// TwinCAT 3 PLC project MRA_LIB
// Title: MRA_LIB
// Company: MRA Solutions
// ProjectVersion: 1.0.5
// ProgramVersion: 3.1.4023.0
// libraries:
//   Tc2_EIB, * (Beckhoff Automation GmbH)
//   Tc2_IoFunctions, * (Beckhoff Automation GmbH)
//   Tc2_ModbusRTU, * (Beckhoff Automation GmbH)
//   Tc2_Standard, * (Beckhoff Automation GmbH)
//   Tc2_System, * (Beckhoff Automation GmbH)
//   Tc2_Utilities, * (Beckhoff Automation GmbH)
//   Tc3_IotBase, * (Beckhoff Automation GmbH)
//   Tc3_IotCommunicator, * (Beckhoff Automation GmbH)
//   Tc3_JsonXml, * (Beckhoff Automation GmbH)
//   Tc3_Module, * (Beckhoff Automation GmbH)
// project tree:
//   MRA/00_DUT/ Klappe_ST.TcDUT
//   MRA/00_GVL/ st_REAL_RRVALUE.TcDUT
//   MRA/00_SYSTEM/ fb_ADS_TIME.TcPOU, fb_BLINKER.TcPOU, fb_DEVICE_RESET.TcPOU
//   MRA/01_FUNKTIONEN/BUS/KNX/ STRING_TO_EIB_GRP_ADDR.TcPOU
//   MRA/01_FUNKTIONEN/MATH/ f_Scale.TcPOU
//   MRA/01_FUNKTIONEN/MQTT/ fb_MQTTSUB.TcPOU, f_MQTTPUB.TcPOU
//   MRA/02_FUNKTIONS_BAUSTEINE/Aggregate/ fb_Klappe.TcPOU, fb_Pumpe.TcPOU, fb_Pumpe_stetig.TcPOU, fb_Ventil_stetig.TcPOU
//   MRA/02_FUNKTIONS_BAUSTEINE/BUS/KNX/ KNX_BOOL_READ_WRITE.TcPOU, KNX_REAL_READ_WRITE.TcPOU
//   MRA/02_FUNKTIONS_BAUSTEINE/BUS/ModBus/ FB_MODBUS_DEVICE.TcPOU
//   MRA/02_FUNKTIONS_BAUSTEINE/MASCHIENENBAU/ fb_Drehzahl.TcPOU
//   MRA/02_FUNKTIONS_BAUSTEINE/Testing/Aggregate/ fb_IBN_Pumpe.TcPOU, fb_IBN_Ventil.TcPOU, fb_IBN_Ventil_ohne_Log.TcPOU
//   MRA/02_FUNKTIONS_BAUSTEINE/Testing/ fb_Log.TcPOU
//   MRA/02_FUNKTIONS_BAUSTEINE/Visualisierung/ fb_Zeitprogramm.TcPOU
//   MRA/03_BSP_PRG/06_KNX/ KNX.TcPOU (excluded from build)
//   MRA/04_RRVALUE/ fb_REAL_RRVALUE.TcPOU
//   MRA/ MAIN.TcPOU
//   / PlcTask.TcTTO
// real-time tasks:
//   TASK PlcTask: cycle T#1ms, priority 20, ADS port 350

CONFIGURATION MRA_LIB
    RESOURCE PLC ON TwinCAT3
        TASK PlcTask(INTERVAL := T#1ms, PRIORITY := 20);
        PROGRAM MAIN WITH PlcTask : MAIN;
    END_RESOURCE
END_CONFIGURATION

// ---- MRA/00_DUT/Klappe_ST.TcDUT
TYPE Klappe_ST :
STRUCT
	BSZ 			:REAL;
	Y_OG			:REAL;
	Y_UG			:REAL;
	V_STELL		:REAL;
	RM_X			:REAL;
	V_SB			:BYTE;		(*~	(SV_Import: true)				(SV_VariableDescription: Betriebsart HAND AUTO)			(SV_Alarm: False)		(SV_Log: True)	 (SV_Command: True)*)
	V_ST			:BYTE;		(*~	(SV_Import: true)				(SV_VariableDescription:Betriebsart Auf Zu)				(SV_Alarm: False)		(SV_Log: True)	 (SV_Command: True)*)
	Status 			:BYTE;		(*~	(SV_Import: true)				(SV_VariableDescription:Status)				(SV_Alarm: False)		(SV_Log: True)	 (SV_Command: False)*)
	(*Bit 0 = Offen / Bit 1 = Störung /  Bit 2 = geschlossen  / Bit 3 = HAND / Bit 4 = Fahrbewegung / Bit 5 = Sperre / Bit 6 = LVB    / Bit 7 = Antrieb angesteuert *)
	BLOCK_EIN		:BOOL;
	NOTB			:BOOL;
	TA_P			:BOOL;
	TA_V			:BOOL;
	TA_G			:BOOL;
	RM				:BOOL;
	RM_AUF			:BOOL;		(*~	(SV_Import: true)				(SV_VariableDescription:Rückmeldung offen)				(SV_Alarm: False)		(SV_Log: True)	 (SV_Command: false)*)
	RM_ZU			:BOOL;		(*~	(SV_Import: true)				(SV_VariableDescription:Rückmeldung geschlossen)		(SV_Alarm: False)		(SV_Log: True)	 (SV_Command: false)*)
	RM_ST1			:BOOL;
	RM_ST2			:BOOL;
	RM_ST3			:BOOL;
	STOE_RM		:BOOL;		(*~	(SV_Import: true)				(SV_VariableDescription:Störung Rückmeldung)			(SV_Alarm: True)		(SV_Log: True)	 (SV_Command: false)*)
	STOE_MS		:BOOL;		(*~	(SV_Import: true)				(SV_VariableDescription:Störung Motorschutz)				(SV_Alarm: True)		(SV_Log: True)	 (SV_Command: false)*)
	STOE_FU		:BOOL;
	STOE_LAUF		:BOOL;
	WART			:BOOL;
	STOE_STB		:BOOL;
	STOE_STROEM:BOOL;
	STOE_FEUCHTE:BOOL;
	Reset_BSZ		:BOOL;
END_STRUCT
END_TYPE

// ---- MRA/00_GVL/st_REAL_RRVALUE.TcDUT
{attribute 'pack_mode' := '1'}
TYPE st_REAL_RRVALUE :
STRUCT
	

	r_in_Value : REAL;
	r_out_Value: REAL;
	
	s_Comment : STRING(1000);
	
	i_Unit : INT;
	//Resolution
	i_Resolution_in_max : INT;
	i_Resolution_in_min : INT;
	i_Resolution_out_max : INT;
	i_Resolution_out_min : INT;	
	//Grenzwert
	r_MaxValue : REAL;
	r_MinValue : REAL;
	b_MaxValue_Reached : BOOL;
	b_MinValue_Reached : BOOL;	
	t_MinMax_Delay : REAL;
	b_Enable_MinMax : BOOL;
	//KNX
	b_KNX_Enable : BOOL;
	s_KNX_Addres : STRING;
	b_KNX_Write_Mode : BOOL;
	
	
END_STRUCT
END_TYPE

// ---- MRA/MAIN.TcPOU
PROGRAM MAIN
VAR
	
IN_TEST_1 AT%I* : BOOL;
		
END_VAR

END_PROGRAM

// ---- MRA/00_SYSTEM/fb_ADS_TIME.TcPOU
FUNCTION_BLOCK fb_ADS_TIME
VAR_INPUT

(*	===============================================================	*)
(*	===						Eingangsvariablen							===		*)
(*	===============================================================	*)

(*	===		BOOL	===	*)


(*	==============================================	*)

(*	===		REAL	===	*)



(*	==============================================	*)

(*	===		STRING	===	*)

	i_AMS_NET_ID	:	STRING :=	''	;

(*	===		WORD	===	*)


(*	==============================================	*)

(*	###################################################################	*)

END_VAR

VAR_OUTPUT

(*	===============================================================	*)
(*	===						Ausgangsvariablen							===		*)
(*	===============================================================	*)

(*	===		DATE_AND_TIME	===	*)

	q_SPS_aktuelle_Uhrzeit	:	DATE_AND_TIME	;
(*	==============================================	*)
(*	===		STRING	===	*)


	Datum				:	STRING			;
	Uhr					:	STRING			;


(*	==============================================	*)
(*	===		WORD	===	*)

	q_SPS_Stunde		:	WORD	;
	q_SPS_Minute		:	WORD	;
	q_SPS_Sekunde		:	WORD	;
	q_SPS_Jahr			:	WORD	;
	q_SPS_Monat		:	WORD	;
	q_SPS_Tag			:	WORD	;
	q_SPS_Wochentag	:	WORD	;

(*	==============================================	*)

(*	###################################################################	*)

END_VAR
VAR

(*	===============================================================	*)
(*	===						interne Variablen								===		*)
(*	===============================================================	*)

	Win_Ce_Zeit		:	TIMESTRUCT	;

	datum_Merker_001	:	STRING	;
	datum_Merker_002	:	STRING	;
	datum_Merker_003	:	STRING	;
	datum_Merker_004	:	STRING	;
	datum_Tag			:	STRING	;
	datum_Monat		:	STRING	;
	datum_Jahr			:	STRING	;
	datum_punkt			:	STRING	:=	'.'	;

	Uhr_Merker_001	:	STRING	;
	Uhr_Merker_002	:	STRING	;
	Uhr_Merker_003	:	STRING	;
	Uhr_Merker_004	:	STRING	;
	Uhr_doppelpunkt	:	STRING		:=	':'	;

	Uhr_Minute	 :	STRING	;
	Uhr_Stunde		:	STRING	;
	Uhr_Sekunde :	STRING	;

(*	###################################################################	*)

(*	===============================================================	*)
(*	===						Zeitvariblen									===		*)
(*	===============================================================	*)

	Intervall_zeit	:	TIME	:=	t#1200ms	;

(*	###################################################################	*)

(*	===============================================================	*)
(*	===						interneBausteine								===		*)
(*	===============================================================	*)


	WinCE_Uhrzeit 		: 	NT_GetTime		;
	lese_interval	: 	TON	;
(*	###################################################################	*)

(*	###################################################################	*)
(*	###################################################################	*)
(*	###################################################################	*)
END_VAR

(*	=================================================	*)
(*	===						Uhrzeitauslesen		    		 ===	*)
(*	=================================================	*)

lese_interval(
	PT	:=			Intervall_zeit,
	IN	:=	NOT	lese_interval.Q
	);

(*	=================================================	*)

WinCE_Uhrzeit		(
(*	----------------------------------------------	*)
(*	Eingaenge	*)
	NETID:=i_AMS_NET_ID ,
	START:=lese_interval.Q ,
(*	Ausgaenge	*)
	TIMESTR=>Win_Ce_Zeit
	 );

(*  ###################################################	*)

(*	=================================================	*)
(*	===			Zeituebergabe an Panel fuer VISU	    		 ===	*)
(*	=================================================	*)

q_SPS_Stunde		:=	Win_Ce_Zeit.wHour			;
q_SPS_Minute		:=	Win_Ce_Zeit.wMinute		;
q_SPS_Sekunde		:=	Win_Ce_Zeit.wSecond		;
q_SPS_Jahr			:=	Win_Ce_Zeit.wYear			;
q_SPS_Monat		:=	Win_Ce_Zeit.wMonth			;
q_SPS_Tag			:=	Win_Ce_Zeit.wDay			;
q_SPS_Wochentag	:=	Win_Ce_Zeit.wDayOfWeek	;



q_SPS_aktuelle_Uhrzeit	:=	SYSTEMTIME_TO_DT
	(	Win_Ce_Zeit	)	;

(*  ###################################################	*)

datum_Tag 		:=	WORD_TO_STRING	(Win_Ce_Zeit.wDay		)	;
datum_Monat 	:=	WORD_TO_STRING	(Win_Ce_Zeit.wMonth		)	;
datum_Jahr 		:=	WORD_TO_STRING	(Win_Ce_Zeit.wYear			)	;

Uhr_Stunde 		:=	WORD_TO_STRING	(Win_Ce_Zeit.wHour		)	;
Uhr_Minute 		:=	WORD_TO_STRING	(Win_Ce_Zeit.wMinute	)	;
Uhr_Sekunde 	:=	WORD_TO_STRING	(Win_Ce_Zeit.wSecond	)	;

datum_Merker_001:= CONCAT	(	datum_Tag			,	datum_punkt		)	;
datum_Merker_002:= CONCAT	(	datum_Merker_001	,	datum_Monat	)	;
datum_Merker_003:=CONCAT	(	datum_Merker_002	,	datum_punkt		)	;
datum_Merker_004:=CONCAT	(	datum_Merker_003	,	datum_Jahr		)	;

datum	:=	datum_Merker_004	;


Uhr_Merker_001:= CONCAT	(	Uhr_Stunde			,	Uhr_doppelpunkt		)	;
Uhr_Merker_002:= CONCAT	(	Uhr_Merker_001		,	Uhr_Minute	)	;
Uhr_Merker_003:=CONCAT	(	Uhr_Merker_002		,	Uhr_doppelpunkt		)	;
Uhr_Merker_004:=CONCAT	(	Uhr_Merker_003		,	Uhr_Sekunde		)	;

Uhr	:=	Uhr_Merker_004	;

(*  ###################################################	*)
(*  ###################################################	*)
(*  ###################################################	*)

END_FUNCTION_BLOCK

// ---- MRA/00_SYSTEM/fb_BLINKER.TcPOU
FUNCTION_BLOCK fb_BLINKER
VAR_INPUT
		///BLINKER///
	bEnable: BOOL;									(*Enable*)
	tImpZeit: TIME;									(*Impulszeit*)
	tPauZeit: TIME;									(*Pausezeit*)
	bStartTyp: BOOL;								(*Start 0=Impuls, 1=Pause*)

	


END_VAR
VAR_OUTPUT
	
	bFreigabe: BOOL;								(*Freigabe Ausgang*)
	tOut: BOOL;											(*Timer Ausgang*)

END_VAR
VAR
	
	flStart: R_TRIG;								(*Start - Flanke*)
	tImpTakt: TON;									(*Impuls Timer*)
	tPauTakt: TON;		

END_VAR



(*Enable*)
IF bEnable = TRUE THEN

	(*Start mit Impuls/Pause*)
	flStart(CLK := bEnable);
	IF flStart.Q = TRUE THEN
		tOut := NOT bStartTyp;
	END_IF

	(*NULL-Zeiten abfragen*)
	IF (tImpZeit > T#0s) AND (tPauZeit > T#0s) THEN

		(*Impuls Takt*)
		tImpTakt(IN := tOut, PT := tImpZeit);
		IF tImpTakt.Q = TRUE THEN
			tOut := FALSE;
		END_IF

		(*Pause Takt*)
		tPauTakt(IN := NOT tOut, PT := tPauZeit);
		IF tPauTakt.Q = TRUE THEN
			tOut := TRUE;
		END_IF

		(*Ausgang*)
		bFreigabe := tOut;

	ELSE

		(*Ausgang*)
		bFreigabe := FALSE;

	END_IF

ELSE

	(*Timer resetieren*)
	tImpTakt.IN := FALSE;
	tImpTakt.PT := T#0s;
	tPauTakt.IN := FALSE;
	tPauTakt.PT := T#0s;

	(*Ausgang*)
	bFreigabe := FALSE;

END_IF

END_FUNCTION_BLOCK

// ---- MRA/00_SYSTEM/fb_DEVICE_RESET.TcPOU
FUNCTION_BLOCK fb_DEVICE_RESET //Dieser FB setzt, anhand des Status des jeweiligen Gerätes (Device ID), jeweils beim erstmaligen überschreiben von Device Status > 0 und nach ablaufen des "DELAY_BETWEEN_RESETS" eine online Reset (Gleich wie über das Kontext Menü bei Rechtsklick auf ein Gerät)
VAR_INPUT
	CX_Status :UINT;
	DEVICEID : UINT;							
	DELAY_BETWEEN_RESETS : TIME := T#10M;	//Zeitintervall zwischen den Rests sollt der status noch 0 werden
	QUIT : BOOL;							//Quttiertaster
	AUTO_RESET_ACTIV : BOOL;				//Freigabe des Autorestieren nach jedem Zeit intervall		
END_VAR
VAR_OUTPUT
	Stoerung_CX : BOOL;						//Wird true bei CX Status größer 0 nach 10 Sekunden
	LOCAL_AMS_NET_ID : STRING;				//AMS Net ID des CX
END_VAR
VAR
	FB_GETLOCALAMSNETID: FB_GetLocalAmsNetId;
	fb_IOF_DeviceReset : IOF_DeviceReset;

	
	TON_KALTSTART: TON;
	TON_CX_Status: TON;
	
	RESET_KBUS: BOOL;
	
	fb_BLINKER : fb_BLINKER;
	
END_VAR



TON_KALTSTART(IN := TRUE, PT := T#2S);

FB_GETLOCALAMSNETID(
	bExecute:= TON_Kaltstart.Q, 
	tTimeOut:= T#500MS);

TON_CX_Status(IN:= CX_Status > 0 , PT:=T#1M , Q=> Stoerung_CX);
	
 fb_BLINKER(
	bEnable:= Stoerung_CX AND RESET_KBUS,
	tImpZeit:= T#5S,
	tPauZeit:= DELAY_BETWEEN_RESETS,
	bStartTyp:= 1,
	tOut => RESET_KBUS	);
	
fb_IOF_DeviceReset(
	NETID:= FB_GETLOCALAMSNETID.AddrString, 
	DEVICEID:= DEVICEID, 
	RESET:= RESET_KBUS OR  QUIT, 
	TMOUT:= T#500MS);

END_FUNCTION_BLOCK

// ---- MRA/01_FUNKTIONEN/BUS/KNX/STRING_TO_EIB_GRP_ADDR.TcPOU
FUNCTION STRING_TO_EIB_GRP_ADDR : EIB_GROUP_ADDR
VAR_INPUT
	GRUPPENADRESSE : STRING;
END_VAR
VAR
	LENGHT: INT;	
	MAIN : BYTE;
	SUBMAIN: BYTE;
	NUMBER: BYTE;	
	GRUPPENADRESSE_BUFFER: STRING(255);
	GRUPPENADRESSE_BUFFER_2: STRING(255);
END_VAR


LENGHT := FIND(GRUPPENADRESSE , '.');


MAIN := STRING_TO_BYTE(LEFT(GRUPPENADRESSE, LENGHT));

CASE LENGHT OF	
	2: GRUPPENADRESSE_BUFFER := DELETE(GRUPPENADRESSE , 2,1);
	3: GRUPPENADRESSE_BUFFER := DELETE(GRUPPENADRESSE , 3,1);
	4: GRUPPENADRESSE_BUFFER := DELETE(GRUPPENADRESSE , 4,1);
END_CASE

LENGHT := FIND(GRUPPENADRESSE_BUFFER , '.');

SUBMAIN := STRING_TO_BYTE(LEFT(GRUPPENADRESSE_BUFFER, LENGHT));

CASE LENGHT OF	
	2: GRUPPENADRESSE_BUFFER_2 := DELETE(GRUPPENADRESSE_BUFFER , 2,1);
	3: GRUPPENADRESSE_BUFFER_2 := DELETE(GRUPPENADRESSE_BUFFER , 3,1);
	4: GRUPPENADRESSE_BUFFER_2 := DELETE(GRUPPENADRESSE_BUFFER , 4,1);
END_CASE


NUMBER := STRING_TO_BYTE(GRUPPENADRESSE_BUFFER_2);

STRING_TO_EIB_GRP_ADDR.MAIN := MAIN;
STRING_TO_EIB_GRP_ADDR.SUB_MAIN := SUBMAIN;
STRING_TO_EIB_GRP_ADDR.NUMBER := NUMBER;

END_FUNCTION

// ---- MRA/01_FUNKTIONEN/MATH/f_Scale.TcPOU
FUNCTION f_Scale : REAL
VAR_INPUT
	input : REAL;
	input_min		:REAL;
	imput_max	:REAL;
	output_min		:REAL;
	output_max	:REAL;
END_VAR

IF (imput_max-input_min) <> 0 THEN
	f_Scale:= (input - input_min)*(output_max-output_min)/(imput_max-input_min)+output_min;
END_IF

IF f_Scale < output_min THEN
	f_Scale:=output_min;
ELSIF f_Scale > output_max THEN
	f_Scale := output_max;
END_IF

END_FUNCTION

// ---- MRA/01_FUNKTIONEN/MQTT/fb_MQTTSUB.TcPOU
FUNCTION_BLOCK fb_MQTTSUB
VAR_INPUT	
	MqttClient : FB_IotMqttClient;
	sTopic : STRING;
END_VAR
VAR_IN_OUT	
	MessageQueue : FB_IotMqttMessageQueue;
END_VAR
VAR_OUTPUT
	sValue : STRING;
END_VAR
VAR
	Message : FB_IotMqttMessage;
END_VAR

MqttClient.Subscribe(sTopic:=sTopic, eQoS:=TcIotMqttQos.AtMostOnceDelivery);

IF MessageQueue.nQueuedMessages > 0 THEN
  
	 IF MessageQueue.Dequeue(fbMessage:=Message) THEN	
		
        IF Message.CompareTopic(sTopic:=sTopic) THEN
            Message.GetPayload(pPayload:=ADR(sValue), nPayloadSize:=SIZEOF(sValue), bSetNullTermination:=FALSE);
	 	END_IF	
		
	END_IF
END_IF

END_FUNCTION_BLOCK

// ---- MRA/01_FUNKTIONEN/MQTT/f_MQTTPUB.TcPOU
FUNCTION f_MQTTPUB : BOOL
VAR_INPUT
	
		MqttClient: FB_IotMqttClient;		
		sTopic : STRING;
		sValue : STRING(3000);

END_VAR
VAR
	sPayloadPub: STRING;
END_VAR

        MqttClient.Publish(    sTopic:= sTopic, 
			                   pPayload:= ADR(sValue), nPayloadSize:= LEN2(ADR(sValue)), 
                               eQoS:= TcIotMqttQos.AtMostOnceDelivery, bRetain:= FALSE, bQueue:= FALSE );

END_FUNCTION

// ---- MRA/02_FUNKTIONS_BAUSTEINE/Aggregate/fb_Klappe.TcPOU
FUNCTION_BLOCK fb_Klappe
(*Klappe - AUF/ZU [1DO] mit Motorschutzschalter*)																


VAR_INPUT
	DDC	:BOOL;	(* 	DDC Betrieb	*)
	FRG	:BOOL;	(* 	Freigabe		*)
	P_HA	:BOOL;	(* 	Panel H/A		*)
	AUTO_AUF	:BOOL;	(* 		*)
	QUITT	:BOOL;	(* 	Störquittierung				*)
	RM_AUF	:BOOL;	(* 	offen	*)
	RM_ZU	:BOOL;	(* 	geschlossen	*)
	BLOCK	:BOOL;	(* 	Blockierschutz	*)
	T_BLOCK	:TIME;	(* 	Aktivierungszeit Blockierschutz	*)
	T_RM	:TIME;	(* 	Rückmeldefehler Zeit		*)
	STOE	:BOOL;	(* 	Störung Motorschutz	*)
	U_IO	:BOOL;	(* 	Spannungsüberwachung			*)
	KONFIG	:BYTE;	(* 	Konfiguration*)
END_VAR

VAR_IN_OUT
	V_SB	:BYTE;	(* 	VISU SB		*)
	V_ST	:BYTE;	(* 	VISU Stufen		*)
	Visu	:Klappe_ST;
END_VAR

VAR_OUTPUT
	NOTB	:BOOL;	(* 	LVB	*)
	TA_P	:BOOL;	(* 	Teilautomatik Panel		*)
	TA_V	:BOOL;	(* 	Teilautomatik VISU		*)
	TA_G	:BOOL;	(* 	Teilautomatik GLT	*)
	S_TA	:BOOL;	(* 	Teilautomatik		*)
	AUF	:BOOL;	(* 	Auf		*)
	STOE_RM	:BOOL;	(* 	Störung Rückmeldung		*)
	STOE_MS	:BOOL;	(* 	Störung Motorschutz	*)
	SA	:BOOL;	(* 	Störung		*)
	BLOCK_EIN	:BOOL;	(* 	Blockierschutz aktiv	*)
	Sperre:BOOL; (*Sperre des Antriebs übergeordnet*)
	RM_offen:BOOL; (*Anzeige Offen Mmeldung*)
	RM_geschlossen:BOOL; (*Anzeige Geschlosen Meldung*)
END_VAR																
VAR
	RMFAuf	:TON;
	RMFZu	:TON;
	QuittRMF	:BOOL;
	Maske	:BYTE;														
	NOTBx	:BOOL;
	TA_Px	:BOOL;														
	TA_Vx	:BOOL;														
	TA_Gx	:BOOL;														
	S_TAx	:BOOL;
	STOE_RM_AUFx	:BOOL;														
	STOE_RM_ZUx	:BOOL;														
	SAx	:BOOL;														
	STOE_MSx	:BOOL;														
	U_IO_Verz	:TON;
	U_IO_X	:BOOL;
	P_AUF	:BOOL;	(* 	Panel Auf	*)
	TON_BLOCK	:TON;
	TP_BLOCK	:TP;
	V_SB_UA_M	:BYTE;														
	V_ST_UA_M	:BYTE;														
	V_STELL_UA_M	:REAL;
	V_SB_M	:BYTE;														
	V_ST_M	:BYTE;														
	V_STELL_M	:REAL;
	
	//MRA
	R_TRIG_RM_AUF : Tc2_Standard.R_TRIG;
	F_TRIG_RM_AUF : Tc2_Standard.F_TRIG;
	R_TRIG_RM_ZU  : Tc2_Standard.R_TRIG;
	F_TRIG_RM_ZU  : Tc2_Standard.F_TRIG;
	ENLAGEN_UW_AUF : BOOL;
	ENLAGEN_UW_ZU : BOOL;
	ANLAGE_HANDBETRIEB: BOOL;
END_VAR

(*Auswertung UA / konventionell*)
IF Visu.V_SB <> V_SB_UA_M THEN
    V_SB_UA_M := Visu.V_SB;
    V_SB_M := Visu.V_SB;
    V_SB := Visu.V_SB;
END_IF;

IF V_SB <> V_SB_M THEN
    V_SB_UA_M := V_SB;
    V_SB_M := V_SB;
    Visu.V_SB := V_SB;
END_IF;

IF Visu.V_ST <> V_ST_UA_M THEN
    V_ST_UA_M := Visu.V_ST;
    V_ST_M := Visu.V_ST;
    V_ST := Visu.V_ST;
END_IF;

IF V_ST <> V_ST_M THEN
    V_ST_UA_M := V_ST;
    V_ST_M := V_ST;
    Visu.V_ST := V_ST;
END_IF;



(*Auswertung VISU/GLT*)
CASE BYTE_TO_INT (V_SB) OF
	1:	TA_Vx	:= TRUE;
		TA_Gx	:= FALSE;
	2:	TA_Vx	:= FALSE;
		TA_Gx	:= TRUE;
	ELSE
		TA_Vx	:= FALSE;
		TA_Gx	:= FALSE;
END_CASE;

(*Initalisierung Stossfreie Umschaltung*)
IF NOT (TA_Gx OR TA_Vx)  THEN
	IF AUF THEN
		V_ST  := 1;
		Visu.V_ST  := 1;
	ELSE
		V_ST := 0;
		Visu.V_ST  := 0;
	END_IF;
END_IF;
IF NOT TA_Px  THEN
	P_AUF  := AUF;
END_IF;

(*Auswertung Panel*)
TA_Px := P_HA;

(*Auswertung Notbetrieb*)
Notbx := NOT DDC;

(*Auswertung Teilautomatik*)
Maske := Konfig AND 2#00010000;
IF Maske = 16 THEN
	S_TAx := TA_Vx OR TA_Gx OR TA_Px;
	ELSE S_TAx := TA_Vx OR TA_Gx OR TA_Px OR Notbx;
END_IF;

R_TRIG_RM_AUF(CLK := RM_AUF);
F_TRIG_RM_AUF(CLK := RM_AUF);
R_TRIG_RM_ZU(CLK := RM_ZU);
F_TRIG_RM_ZU(CLK := RM_ZU);

(*Auswertung Rückmeldefehler*)
IF AUTO_AUF AND R_TRIG_RM_AUF.Q THEN
	ENLAGEN_UW_AUF := TRUE;
ELSIF NOT AUTO_AUF THEN
	ENLAGEN_UW_AUF := FALSE;	
END_IF

IF NOT AUTO_AUF AND R_TRIG_RM_ZU.Q THEN
	ENLAGEN_UW_ZU := TRUE;
ELSIF AUTO_AUF THEN
	ENLAGEN_UW_ZU := FALSE;	
END_IF

IF (ENLAGEN_UW_AUF AND NOT RM_AUF) OR (ENLAGEN_UW_ZU AND NOT RM_ZU)  THEN
	ANLAGE_HANDBETRIEB := TRUE;
ELSIF QUITT AND (((ENLAGEN_UW_AUF AND RM_AUF) OR (ENLAGEN_UW_ZU AND RM_ZU)) OR (NOT ENLAGEN_UW_AUF OR NOT ENLAGEN_UW_ZU))  THEN
	ANLAGE_HANDBETRIEB := FALSE;
END_IF




RMFAuf (IN:=(((RM_AUF XOR AUF) AND DDC) OR Stoe_Rm_AUFx) AND NOT QuittRMF, PT:=T_RM);
RMFZu  (IN:=(((RM_ZU XOR NOT AUF) AND DDC) OR Stoe_Rm_ZUx) AND NOT QuittRMF, PT:=T_RM);
Stoe_Rm_AUFx := RMFAuf.Q OR ANLAGE_HANDBETRIEB;
Stoe_Rm_ZUx := RMFZu.Q OR ANLAGE_HANDBETRIEB;

(*Auswertung Motorschutz*)
Stoe_Msx := (NOT Stoe OR Stoe_Msx) AND NOT (Stoe AND Quitt);

(*Auswertung Störung*)
Maske := Konfig AND 2#00001000;
IF Maske = 8 THEN
	SAx := Stoe_Msx OR (Stoe_Rm_Aufx OR Stoe_Rm_Zux);
	ELSE	SAx := Stoe_Msx OR (Stoe_Rm_Aufx OR Stoe_Rm_Zux);
END_IF;

(*Quittierung Rückmeldefehler*)
QuittRMF := FALSE;
Maske := Konfig AND 2#00000001;
IF Maske = 1 THEN
	IF (Auf AND Rm_Auf OR NOT Auf AND RM_Zu) AND (Stoe_Rm_Aufx OR Stoe_Rm_Zux) AND Quitt THEN
		QuittRMF := TRUE;
	END_IF;
	ELSE IF (Stoe_Rm_Aufx OR Stoe_Rm_Zux) AND Quitt THEN
		QuittRMF := TRUE;
	END_IF;
END_IF;

(*Ansteuerung Antrieb*)
IF FRG AND DDC AND NOT Stoe_Msx THEN
	Auf := Auto_Auf;
	IF TA_Gx OR TA_Vx THEN
		Maske := 2#00000001;
		Auf := BYTE_TO_BOOL (Maske AND V_ST);
	END_IF;
	IF TA_Px THEN
		Auf := P_Auf;
	END_IF;
		Auf := Auf OR  TP_BLOCK.Q;	(*Blockierschutz*);
	IF (Stoe_Rm_Aufx OR Stoe_Rm_Zux) THEN	(*Bei Rückmeldefehler Antrieb = Ein || Antrieb = Aus || Antrieb = Auto*)
		Maske := Konfig AND 2#00000110;
		IF Maske = 4 THEN
			Auf := Auf;
			ELSE IF Maske = 2 THEN
				Auf := TRUE;
				ELSE Auf := FALSE;
			END_IF;
		END_IF;
	END_IF;




	(*Blockierschutz*)
	TON_BLOCK (IN:= BLOCK AND NOT Auf, PT:=T_BLOCK);
	TP_BLOCK (IN:= TON_BLOCK.Q, PT:= T#10s);
	IF TP_BLOCK.Q THEN
		AUF := TRUE;
	END_IF;

	BLOCK_EIN := TP_BLOCK.Q;

	ELSE AUF := FALSE;
END_IF;
(*Meldeunterdrückung*)
U_IO_Verz(IN:=U_IO, PT:=T#5s);
U_IO_X := U_IO_Verz.Q;
IF U_IO_X THEN
	NOTB	:=	NOTBx	;
	TA_P	:=	TA_Px	;
	TA_V	:=	TA_Vx	;
	TA_G	:=	TA_Gx	;
	S_TA	:=	S_TAx	;
	STOE_RM	:=	(Stoe_Rm_Aufx OR Stoe_Rm_Zux)	;
	STOE_MS	:=	STOE_MSx	;
	SA	:=	SAx	;
END_IF;

RM_offen:= RM_AUF;
RM_geschlossen:= RM_ZU;


Sperre:=NOT FRG;

VISU.NOTB    :=    NOTB;
VISU.TA_P    :=    TA_P;
VISU.TA_V    :=    TA_V;
VISU.TA_G    :=    TA_G;

VISU.RM		:=    FALSE;
VISU.RM_AUF	:=	RM_AUF;
VISU.RM_ZU	:=	RM_ZU;
VISU.RM_ST1	:=	FALSE;
VISU.RM_ST2	:=	FALSE;
VISU.RM_ST3	:=	FALSE;

VISU.STOE_RM		:=    STOE_RM;
VISU.STOE_MS		:=    STOE_MS;
VISU.STOE_FU	 	:=    FALSE;
VISU.Stoe_Lauf		:=    FALSE;
VISU.Wart			:=	FALSE;
VISU.STOE_STB	:=	FALSE;
VISU.STOE_STROEM	:=	FALSE;
VISU.STOE_FEUCHTE	:=	FALSE;

VISU.Y_OG			:=	0;
VISU.Y_UG			:=	0;
VISU.RM_X  		:=    0;

Visu.Status.0:=RM_AUF;
Visu.Status.1:=SA;
Visu.Status.2:=RM_ZU;
Visu.Status.3:=S_TA;
Visu.Status.4:=NOT RM_AUF AND NOT RM_ZU;
Visu.Status.5:=Sperre;
Visu.Status.6:=NOT NOTB;
Visu.Status.7:=AUF;

END_FUNCTION_BLOCK

// ---- MRA/02_FUNKTIONS_BAUSTEINE/Aggregate/fb_Pumpe.TcPOU
FUNCTION_BLOCK fb_Pumpe
(*Pumpe*)

VAR_INPUT
	DDC	:BOOL;	(* 	DDC Betrieb	*)
	FRG	:BOOL;	(* 	Freigabe	*)
	P_HA	:BOOL;	(* 	Panel H/A	*)
	AUTO	:BOOL;	(* 	Auto Betrieb	*)
	QUITT	:BOOL;	(* 	Störquittierung	*)
	RM		:BOOL;	(* 	RM Betrieb	*)
	T_RM	:TIME;	(* 	Rückmeldefehler Zeit	*)
	STOE	:BOOL;	(* 	Störung Motorschutz	*)
	REP	:BOOL;	(* 	Rep.-Schalter	*)	
	FROST	:BOOL;	(* 	Frostschutz	*)
	BLOCK	:BOOL;	(* 	Blockierschutz	*)
	T_BLOCK	:TIME;	(* 	Aktivierungszeit Blockierschutz	*)
	U_IO	:BOOL;	(* 	Spannungsüberwachung	*)
	KONFIG	:BYTE;	(*	
						2#00010000 Auswertung Teilautomatik
						2#00001000 Auswertung Störung
						2#00000100 Bei Rückmeldefehler Antrieb = Auto
						2#00000010 Bei Rückmeldefehler Antrieb = Ein
						2#00000001 Quittierung Rückmeldefehler
						*)
	Reset_BSZ:BOOL;	(* 	Rücksetzen BSZ	*)
	Nachlaufzeit		:TIME := T#5S; (* 	Nachlaufzeit der Pumpe	*)
END_VAR

VAR_IN_OUT
	V_SB	:BYTE;		(* 	VISU SB*)
	V_ST	:BYTE;		(* 	VISU Stufen*)
	BSZ:REAL;			(* 	Betriebsstundenzähler*)

END_VAR

VAR_OUTPUT
	NOTB	:BOOL;	(* 	LVB	*)
	TA_P	:BOOL;	(* 	Teilautomatik Panel	*)
	TA_V	:BOOL;	(* 	Teilautomatik VISU	*)
	TA_G	:BOOL;	(* 	Teilautomatik GLT	*)
	S_TA	:BOOL;	(* 	Teilautomatik	*)
	EIN	:BOOL;	(* 	Betrieb	*)
	STOE_RM	:BOOL;	(* 	Störung Rückmeldung	*)
	STOE_MS	:BOOL;	(* 	Störung Motorschutz	*)
	STOE_FROST	:BOOL;	(* 	Störung Frostschutz	*)
	BLOCK_EIN	:BOOL;	(* 	Blockierschutz aktiv	*)
	WART	:BOOL;	(* 	Reparaturschalter	*)
	SA	:BOOL;	(* 	Störung	*)
	Betrieb:BOOL;	(* 	Betriebsmeldung	*)
	Sperre:BOOL;(* 	Sperre Antrieb (Keine Freigabe)	*)
END_VAR
VAR
	RMF	:TON;
	QuittRMF	:BOOL;
	Maske	:BYTE;
	NOTBx	:BOOL;														
	TA_Px	:BOOL;														
	TA_Vx	:BOOL;														
	TA_Gx	:BOOL;
	S_TAx	:BOOL;														
	STOE_RMx	:BOOL;														
	STOE_MSx	:BOOL;
	SAx	:BOOL;
	Wartx	:BOOL;														
	Stoe_Laufx	:BOOL;
	Stoe_Frostx	:BOOL;
	TON_BLOCK	:TON;
	TP_BLOCK	:TP;
	U_IO_Verz	:TON;
	U_IO_X	:BOOL;
	BSZ_Pumpe: FB_ALB_BSZ;
	TOF_AUSVZ	:TOF;

	Wartung:REAL;
	Intervall_WA:REAL:=0;
	P_EIN	:BOOL;	(* 	Panel Ein*)
	V_SB_UA_M	:BYTE;														
	V_ST_UA_M	:BYTE;
	V_STELL_UA_M	:REAL;
	V_SB_M	:BYTE;														
	V_ST_M	:BYTE;
	V_STELL_M	:REAL;
END_VAR

(*Auswertung UA / konventionell*)


IF V_SB <> V_SB_M THEN
    V_SB_UA_M := V_SB;
    V_SB_M := V_SB;
END_IF;




IF V_ST <> V_ST_M THEN
    V_ST_UA_M := V_ST;
    V_ST_M := V_ST;
END_IF;


(*Auswertung VISU/GLT*)
CASE BYTE_TO_INT (V_SB) OF
	1:	TA_Vx	:= TRUE;
		TA_Gx	:= FALSE;
	2:	TA_Vx	:= FALSE;
		TA_Gx	:= TRUE;
	ELSE
		TA_Vx	:= FALSE;
		TA_Gx	:= FALSE;
END_CASE;

(*Initalisierung Stossfreie Umschaltung*)
IF NOT (TA_Gx OR TA_Vx)  THEN
	IF EIN THEN
		V_ST  := 1;

	ELSE
		V_ST := 0;

	END_IF;
END_IF;
IF NOT TA_Px  THEN
	P_EIN  := EIN;
END_IF;

(*Auswertung Panel*)
TA_Px := P_HA;

(*Auswertung Notbetrieb*)
Notbx := NOT DDC;

(*Auswertung Teilautomatik*)
Maske := Konfig AND 2#00010000;
IF Maske = 16 THEN
	S_TAx := TA_Vx OR TA_Gx OR TA_Px;
	ELSE S_TAx := TA_Vx OR TA_Gx OR TA_Px OR Notbx;
END_IF;

(*Auswertung Rückmeldefehler*)
RMF(IN:=(((Ein XOR Rm) AND DDC) OR Stoe_Rmx) AND NOT QuittRMF, PT:=T_RM);
Stoe_Rmx := RMF.Q;

(*Auswertung Motorschutz*)
Stoe_Msx := (NOT Stoe OR Stoe_Msx) AND NOT (Stoe AND Quitt);

(*Auswertung Frostschutz*)
Stoe_Frostx := (NOT Frost OR Stoe_Frostx) AND NOT (Frost AND Quitt);

(*Auswertung Störung*)
Maske := Konfig AND 2#00001000;
IF Maske = 8 THEN
	SAx := Stoe_Msx OR Stoe_Rmx OR Stoe_Laufx OR Wartx;
	ELSE	SAx := Stoe_Msx OR Stoe_Rmx OR Stoe_Laufx;
END_IF;

(*Auswertung Rep.-Schalter*)
IF Maske = 8 THEN
	Wartx := NOT REP OR Wartx AND NOT Quitt;
	ELSE Wartx := NOT REP;
END_IF;

(*Quittierung Rückmeldefehler*)
QuittRMF := FALSE;
Maske := Konfig AND 2#00000001;
IF Maske = 1 THEN
	IF (Ein = Rm) AND Stoe_Rmx AND Quitt THEN
		QuittRMF := TRUE;
	END_IF;
	ELSE IF Stoe_Rmx AND Quitt THEN
		QuittRMF := TRUE;
	END_IF;
END_IF;

(*Nachlaufzeit Pumpe *)

TOF_AUSVZ(IN:=Auto , PT:=Nachlaufzeit, Q=> , ET=> );

(*Ansteuerung Antrieb*)
IF FRG AND DDC AND NOT Stoe_Msx AND NOT Wartx THEN
	Ein := TOF_AUSVZ.Q;
	IF TA_Gx OR TA_Vx THEN
		Maske := 2#00000001;
		Ein := BYTE_TO_BOOL (Maske AND V_ST);
	END_IF;
	IF TA_Px THEN
		Ein := P_Ein;
	END_IF;
	Ein := Ein OR TP_BLOCK.Q;	(*Blockierschutz*)
	IF Stoe_Rmx THEN	(*Bei Rückmeldefehler Antrieb = Ein || Antrieb = Aus || Antrieb = Auto*)
		Maske := Konfig AND 2#00000110;
		IF Maske = 4 THEN
			Ein := Ein;
			ELSE IF Maske = 2 THEN
				Ein := TRUE;
				ELSE Ein := FALSE;
			END_IF;
		END_IF;
	END_IF;

	IF STOE_Frost THEN	(*Übersteuerung Frostschutz*)
		Ein := TRUE;
	END_IF;

	(*Blockierschutz*)
	TON_BLOCK (IN:= BLOCK AND NOT EIN, PT:=T_BLOCK);
	TP_BLOCK (IN:= TON_BLOCK.Q, PT:= T#5m);
	IF TP_BLOCK.Q THEN
		Ein := TRUE;
	END_IF;

	BLOCK_EIN := TP_BLOCK.Q;

	ELSE Ein := FALSE;
END_IF;

(*Meldeunterdrückung*)
U_IO_Verz(IN:=U_IO, PT:=T#5s);
U_IO_X := U_IO_Verz.Q;
IF U_IO_X THEN
	NOTB	:=	NOTBx	;
	TA_P	:=	TA_Px	;
	TA_V	:=	TA_Vx	;
	TA_G	:=	TA_Gx	;
	S_TA	:=	S_TAx	;
	STOE_RM	:=	STOE_RMx	;
	STOE_MS	:=	STOE_MSx	;
	SA	:=	SAx	;
	Wart	:=	Wartx	;
	STOE_FROST	:= Stoe_Frostx;
END_IF;

Betrieb:=RM;
Sperre:=NOT FRG;



(****************Betriebsstundenzaehler*)

BSZ_Pumpe(
	RM:= RM,
	Reset:=VISU.Reset_BSZ OR Reset_BSZ,
	INTERVALL:=Intervall_WA ,
	WERT:= BSZ,
	WARTUNG:= Wartung);

END_FUNCTION_BLOCK

// ---- MRA/02_FUNKTIONS_BAUSTEINE/Aggregate/fb_Pumpe_stetig.TcPOU
FUNCTION_BLOCK fb_Pumpe_stetig
(*Antrieb mit FU*)

VAR_INPUT
	DDC	:BOOL;	(* 	DDC Betrieb	*)
	HAND_FU	:BOOL;	(*	Handbetrieb FU	*)
	FRG	:BOOL;	(* 	Freigabe	*)
	P_HA	:BOOL;	(* 	Panel H/A	*)
	AUTO	:BOOL;	(* 	Auto Betrieb	*)
	AUTO_STELL	:REAL;	(* 	Auto Stellbefehl	*)
	QUITT	:BOOL;	(* 	Störquittierung	*)
	RM	:BOOL;	(* 	RM Betrieb FU	*)
	T_RM	:TIME;	(* 	Rückmeldefehler Zeit	*)
	STOE	:BOOL;	(* 	Störung Motorschutz	*)
	SA_FU	:BOOL;	(* 	Störung FU	*)
	REP	:BOOL;	(* 	Rep.-Schalter	*)
	LAUF	:BOOL;	(* 	Laufüberwachung	*)
	T_LAUF	:TIME;	(* 	Laufüberwachung Zeit	*)
	RM_Y	:INT;	(*	Rückmeldung	*)
	Y_OG	:REAL;	(*	Obergrenze	*)
	Y_UG	:REAL;	(*	Untergrenze	*)
	U_IO	:BOOL;	(* 	Spannungsüberwachung	*)
	KONFIG	:BYTE;	(* 	Konfiguration	*)
	Reset_BSZ:BOOL;	(* 	Rücksetzen BSZ	*)
END_VAR					
VAR_IN_OUT
	V_SB	:BYTE;	(* 	VISU SB	*)
	V_ST	:BYTE;	(* 	VISU Stufen	*)
	V_STELL	:REAL;	(* 	VISU Stellbefehl	*)
	BSZ:REAL;			(* 	Betriebsstundenzähler*)
END_VAR

VAR_OUTPUT
	NOTB	:BOOL;	(* 	LVB	*)
	TA_P	:BOOL;	(* 	Teilautomatik Panel	*)
	TA_V	:BOOL;	(* 	Teilautomatik VISU	*)
	TA_G	:BOOL;	(* 	Teilautomatik GLT	*)
	S_TA	:BOOL;	(* 	Teilautomatik	*)
	EIN	:BOOL;		(* 	Betrieb FU	*)
	Betrieb:BOOL;	(* 	Betriebsmeldung	*)
	RM_X	:REAL;	(*	Rückmeldung	*)
	Y	:REAL;		(*	Stellsignal	*)
	Y_OUT	:INT;	(*	Stellsignal	*)
	STOE_RM	:BOOL;	(* 	Störung Rückmeldung	*)
	STOE_MS	:BOOL;	(* 	Störung Motorschutz	*)
	STOE_FU	:BOOL;	(* 	Störung FU	*)
	STOE_LAUF	:BOOL;	(* 	Störung Laufüberwachung	*)
	WART	:BOOL;	(* 	Reparatur	*)
	SA	:BOOL;	(* 	Störung	*)
	Sperre:BOOL; (*Übergeordnete Sperre Antrieb*)

END_VAR
VAR
	BSZ_Pumpe: FB_ALB_BSZ;
	Wartung:REAL;
	Intervall_WA:REAL:=0;
	P_EIN	:BOOL;	(* 	Panel Ein	*)
	P_STELL	:REAL;	(* 	Panel Stellbefehl	*)
	RMF	:TON;
	LaufZeit	:TON;
	QuittRMF	:BOOL;														
	Maske	:BYTE;														
	NOTBx	:BOOL;
	TA_Px	:BOOL;
	TA_Vx	:BOOL;														
	TA_Gx	:BOOL;
	S_TAx	:BOOL;
	STOE_RMx	:BOOL;														
	STOE_MSx	:BOOL;
	SAx	:BOOL;
	Wartx	:BOOL;														
	Stoe_Laufx	:BOOL;
	Stoe_Fux	:BOOL;
	Yx	:REAL;
	m	:REAL;														
	b	:REAL;														
	U_IO_Verz	:TON;														
	U_IO_X	:BOOL;



	V_SB_UA_M	:BYTE;														
	V_ST_UA_M	:BYTE;
	V_STELL_UA_M	:REAL;														
	V_SB_M	:BYTE;														
	V_ST_M	:BYTE;
	V_STELL_M	:REAL;														
END_VAR

(*Auswertung UA / konventionell*)


IF V_SB <> V_SB_M THEN
    V_SB_UA_M := V_SB;
    V_SB_M := V_SB;
END_IF;



IF V_ST <> V_ST_M THEN
    V_ST_UA_M := V_ST;
    V_ST_M := V_ST;

END_IF;



IF V_STELL <> V_STELL_M THEN
    V_STELL_UA_M := V_STELL;
    V_STELL_M := V_STELL;
 
END_IF;

(*Auswertung VISU/GLT*)
CASE BYTE_TO_INT (V_SB) OF
    1:    	TA_Vx    := TRUE;
      	  	TA_Gx    := FALSE;
    2:    	TA_Vx    := FALSE;
       		TA_Gx    := TRUE;
    ELSE
        TA_Vx    := FALSE;
        TA_Gx    := FALSE;
END_CASE;

(*Auswertung Panel*)
TA_Px := P_HA;

(*Auswertung Notbetrieb*)
Notbx := NOT DDC OR NOT HAND_FU;

(*Initalisierung Stossfreie Umschaltung*)
IF (NOT (TA_Gx OR TA_Vx)) OR TA_Px THEN
    IF EIN THEN
        V_ST  := 1;
        Visu.V_ST := 1;
        ELSE
            V_ST := 0;
         
    END_IF;
    V_STELL := Y;
  
ELSE
    IF V_ST = 0  THEN
        V_STELL := 0;
     
    END_IF;
END_IF;
IF NOT TA_Px  THEN
    P_EIN  := EIN;
    P_STELL := Y;
ELSE
    IF NOT P_EIN THEN
        P_STELL := 0;
    END_IF;
END_IF;

(*Auswertung Teilautomatik*)
Maske := Konfig AND 2#00010000;
IF Maske = 16 THEN
    S_TAx := TA_Vx OR TA_Gx OR TA_Px;
    ELSE S_TAx := TA_Vx OR TA_Gx OR TA_Px OR Notbx;
END_IF;

(*Auswertung Rückmeldefehler*)
RMF(IN:=(((Ein XOR Rm) AND DDC) OR Stoe_Rmx) AND NOT QuittRMF, PT:=T_RM);
Stoe_Rmx := RMF.Q;

(*Auswertung Motorschutz*)
Stoe_Msx := (NOT Stoe OR Stoe_Msx) AND NOT (Stoe AND Quitt);

(*Auswertung Störung FU*)
Stoe_FUx := (NOT SA_FU OR Stoe_FUx) AND NOT (SA_FU AND Quitt);

(*Auswertung Störung*)
Maske := Konfig AND 2#00001000;
IF Maske = 8 THEN
    SAx := Stoe_Msx OR Stoe_Rmx OR Stoe_Laufx OR Wartx OR Stoe_FUx ;
    ELSE    SAx := Stoe_Msx OR Stoe_Rmx OR Stoe_Laufx OR Stoe_FUx ;
END_IF;

(*Auswertung Rep.-Schalter*)
IF Maske = 8 THEN
    Wartx := NOT REP OR Wartx AND NOT Quitt;
    ELSE Wartx := NOT REP;
END_IF;

(*Auswertung Laufüberwachung*)
LaufZeit(IN:=((RM AND NOT Lauf) OR Stoe_Laufx) AND NOT Quitt, PT:= T_Lauf);
Stoe_Laufx := LaufZeit.Q;

(*Quittierung Rückmeldefehler*)
QuittRMF := FALSE;
Maske := Konfig AND 2#00000001;
IF Maske = 1 THEN
    IF (Ein = Rm) AND Stoe_Rmx AND Quitt THEN
        QuittRMF := TRUE;
    END_IF;
    ELSE IF Stoe_Rmx AND Quitt THEN
        QuittRMF := TRUE;
    END_IF;
END_IF;

(*Ansteuerung Antrieb*)
IF FRG AND DDC AND NOT Stoe_Msx AND NOT Wartx AND NOT Stoe_Laufx AND NOT Stoe_FUx THEN
    Ein := Auto;
    IF NOT Auto THEN
        Auto_Stell := 0;
    END_IF;
    m := ((Y_OG - Y_UG) / 100);    (*Steigung*)
    b := Y_UG;                    (*Nulldurchgang*)
    Yx := m * Auto_Stell + b;        (*Geradengleichung*)
    IF TA_Gx OR TA_Vx THEN
        Maske := 2#00000001;
        Ein := BYTE_TO_BOOL (Maske AND V_ST);
        IF V_STELL > Y_OG THEN
            V_STELL := Y_OG;
        END_IF;
        IF V_STELL < Y_UG THEN
            V_STELL := Y_UG;
        END_IF;
        Yx := V_STELL;
    END_IF;
    IF TA_Px THEN
        Ein := P_Ein;
        IF P_STELL > Y_OG THEN
            P_STELL := Y_OG;
        END_IF;
        IF P_STELL < Y_UG THEN
            P_STELL := Y_UG;
        END_IF;
        Yx := P_STELL;
    END_IF;
    IF Stoe_Rmx THEN    (*Bei Rückmeldefehler Antrieb = Ein || Antrieb = Aus || Antrieb = Auto*)
        Maske := Konfig AND 2#00000110;
        IF Maske = 4 THEN
            Ein := Ein;
            Yx := Yx;
            ELSE IF Maske = 2 THEN
                Ein := TRUE;
                Yx := Y_OG;
                ELSE
                    Ein := FALSE;
                    Yx := Y_UG;
            END_IF;
        END_IF;
    END_IF;
ELSE
    Ein := FALSE;
    Yx := Y_UG;
END_IF;

(*Skalierung Ansteuerung*)
IF  (Y_OG - Y_UG) = 0 THEN
    Y_OUT := 0;                                    (*DIV / NULL*)
    ELSE
        m := (32767 / (Y_OG - Y_UG));            (*Steigung*)
        b := Y_UG * m * -1;                        (*Nulldurchgang*)
        Y_OUT := REAL_TO_INT (m * Yx + b);    (*Geradengleichung*)

	(*Ansteuerung gegenläufig*)
	Maske := Konfig AND 2#01000000;
	IF Maske = 64 THEN
		m :=-1;	(*Steigung*)
		b := 32767;
		Y_OUT :=REAL_TO_INT( INT_TO_REAL (Y_OUT) * m + b);
	END_IF;

	(*Ansteuerung 2-10V*)
	Maske := Konfig AND 2#00100000;
	IF Maske = 32 THEN
		m :=0.8;	(*Steigung*)
		b := 0.2 * 32767;
		Y_OUT :=REAL_TO_INT( INT_TO_REAL (Y_OUT) * m + b);
	END_IF;
END_IF;

(*Rückmeldung gegenläufig*)
Maske := Konfig AND 2#01000000;
IF Maske = 64 THEN
	m :=-1;	(*Steigung*)
	b := 32767;
	RM_Y :=REAL_TO_INT( INT_TO_REAL (RM_Y) * m + b);
END_IF;

(*Rückmeldung 2-10V*)
Maske := Konfig AND 2#00100000;
IF Maske = 32 THEN
	m :=1.25;	(*Steigung*)
	b := -0.25 * 32767;
	RM_Y :=REAL_TO_INT( INT_TO_REAL (RM_Y) * m + b);
END_IF;

(*Skalierung Rückmeldung*)
m := ((Y_OG - Y_UG) / 32767);    (*Steigung*)
b := Y_UG;                    (*Nulldurchgang*)
RM_X := m * INT_TO_REAL (RM_Y) + b;        (*Geradengleichung*)
IF RM_X < Y_UG THEN
    RM_X := Y_UG;
END_IF;
IF RM_X > Y_OG THEN
    RM_X := Y_OG;
END_IF;
IF NOT RM THEN
    RM_X := 0;
    Yx := 0;
END_IF;

Y := Yx;
(*Meldeunterdrückung*)
U_IO_Verz(IN:=U_IO, PT:=T#5s);
U_IO_X := U_IO_Verz.Q;
IF U_IO_X THEN
    NOTB    :=    NOTBx    ;
    TA_P    :=    TA_Px    ;
    TA_V    :=    TA_Vx    ;
    TA_G    :=    TA_Gx    ;
    S_TA    :=    S_TAx    ;
    STOE_RM    :=    STOE_RMx    ;
    STOE_MS    :=    STOE_MSx    ;
    STOE_FU    :=    STOE_FUx    ;
    SA    :=    SAx    ;
    Wart    :=    Wartx    ;
    Stoe_Lauf    :=    Stoe_Laufx    ;
END_IF;

Sperre:=NOT FRG;
Betrieb:=RM AND LAUF;

(****************Betriebsstundenzaehler*)

BSZ_Pumpe(
	RM:= Betrieb,
	Reset:=VISU.Reset_BSZ OR Reset_BSZ,
	INTERVALL:=Intervall_WA ,
	WERT:= BSZ,
	WARTUNG:= Wartung);

END_FUNCTION_BLOCK

// ---- MRA/02_FUNKTIONS_BAUSTEINE/Aggregate/fb_Ventil_stetig.TcPOU
FUNCTION_BLOCK fb_Ventil_stetig
(*Ventil-stetig*)																


VAR_INPUT
	DDC	:BOOL;	(* 	DDC Betrieb	*)
	FRG	:BOOL;	(* 	Freigabe			*)
	P_HA	:BOOL;	(* 	Panel H/A	*)
	AUTO_STELL	:REAL;	(* 	Auto Stellbefehl*)
	FROST	:BOOL;	(* 	Frostschutz					*)
	RM_Y	:INT;	(*	Rückmeldung		*)
	QUITT	:BOOL;	(* 	Störquittierung	*)
	T_RM	:TIME;	(* 	Rückmeldefehler Zeit	*)
	Y_OG	:REAL;	(*	Obergrenze	*)
	Y_UG	:REAL;	(*	Untergrenze	*)
	BLOCK	:BOOL;	(* 	Blockierschutz	*)
	T_BLOCK	:TIME;	(* 	Aktivierungszeit Blockierschutz	*)
	U_IO	:BOOL;	(* 	Spannungsüberwachung		*)
	KONFIG	:BYTE;	(* 	Konfiguration	
						2#01000000 Ansteuerung&Rückmeldung Gegenläufig
						2#00100000 Ansteuerung&Rückmeldung 2-10V
						2#00010000 Auswertung Teilautomatik
						2#00001000 Auswertung Störung
						2#00000100 Bei Rückmeldefehler Antrieb = Auto
						2#00000010 Bei Rückmeldefehler Antrieb = Ein
						2#00000001 Quittierung Rückmeldefehler*)
END_VAR
VAR_IN_OUT
	V_SB	:BYTE;	(* 	VISU SB	*)
	V_STELL	:REAL;	(* 	VISU Stellbefehl	*)
END_VAR					

VAR_OUTPUT					
	NOTB	:BOOL;	(* 	LVB	*)
	TA_P	:BOOL;	(* 	Teilautomatik Panel	*)
	TA_V	:BOOL;	(* 	Teilautomatik VISU	*)
	TA_G	:BOOL;	(* 	Teilautomatik GLT	*)
	S_TA	:BOOL;	(* 	Teilautomatik	*)
	Y	:REAL;	(*	Stellsignal	*)
	Y_OUT	:INT;	(*	Stellsignal	*)
	STOE_RM	:BOOL;	(* 	Störung Rückmeldung	*)
	STOE_FROST	:BOOL;	(* 	Störung Frostschutz	*)
	BLOCK_EIN	:BOOL;	(* 	Blockierschutz aktiv	*)
	SA	:BOOL;	(* 	Störung	*)
	RM_X	:REAL;	(*	Rückmeldung	*)
	Sperre:BOOL;(* 	Sperre Ventil (Keine Freigabe)	*)
END_VAR					


VAR
	P_STELL	:REAL;	(* 	Panel Stellbefehl	*)
	RMF	:TON;														
	QuittRMF	:BOOL;														
	Maske	:BYTE;														
	NOTBx	:BOOL;														
	TA_Px	:BOOL;														
	TA_Vx	:BOOL;														
	TA_Gx	:BOOL;														
	S_TAx	:BOOL;														
	STOE_RMx	:BOOL;														
	SAx	:BOOL;														
	Yx	:REAL;														
	m	:REAL;														
	b	:REAL;														
	Stoe_Frostx	:BOOL;														
	BereichOG	:REAL;														
	BereichUG	:REAL;														
	TON_BLOCK	:TON;
	TP_BLOCK	:TP;														
	U_IO_Verz	:TON;														
	U_IO_X	:BOOL;														


	V_SB_UA_M	:BYTE;
	V_ST_UA_M	:BYTE;
	V_STELL_UA_M	:REAL;														
	V_SB_M	:BYTE;														
	V_ST_M	:BYTE;
	V_STELL_M	:REAL;														
END_VAR

(*Auswertung UA / konventionell*)


IF V_SB <> V_SB_M THEN
    V_SB_UA_M := V_SB;
    V_SB_M := V_SB;
END_IF;



IF V_STELL <> V_STELL_M THEN
    V_STELL_UA_M := V_STELL;
    V_STELL_M := V_STELL;
END_IF;


(*Auswertung VISU/GLT*)
CASE BYTE_TO_INT (V_SB) OF
	1:	TA_Vx	:= TRUE;
		TA_Gx	:= FALSE;
	2:	TA_Vx	:= FALSE;
		TA_Gx	:= TRUE;
	ELSE
		TA_Vx	:= FALSE;
		TA_Gx	:= FALSE;
END_CASE;

(*Initalisierung Stossfreie Umschaltung*)
IF NOT (TA_Gx OR TA_Vx)  THEN
	V_STELL := Y;
END_IF;
IF NOT TA_Px  THEN
	P_STELL :=Y;
END_IF;

(*Auswertung Panel*)
TA_Px := P_HA;

(*Auswertung Notbetrieb*)
Notbx := NOT DDC;

(*Auswertung Teilautomatik*)
Maske := Konfig AND 2#00010000;
IF Maske = 16 THEN
	S_TAx := TA_Vx OR TA_Gx OR TA_Px;
	ELSE S_TAx := TA_Vx OR TA_Gx OR TA_Px OR Notbx;
END_IF;

(*Rückmeldung gegenläufig*)
Maske := Konfig AND 2#01000000;
IF Maske = 64 THEN
	m :=-1;	(*Steigung*)
	b := 32767;
	RM_Y :=REAL_TO_INT( INT_TO_REAL (RM_Y) * m + b);
END_IF;

(*Rückmeldung 2-10V*)
Maske := Konfig AND 2#00100000;
IF Maske = 32 THEN
	m :=1.25;	(*Steigung*)
	b := -0.25 * 32767;
	RM_Y :=REAL_TO_INT( INT_TO_REAL (RM_Y) * m + b);
END_IF;

(*Auswertung Rückmeldung*)
m := ((Y_OG - Y_UG)/32767);					(*Steigung*)
b  := Y_UG;										(*Nulldurchgang*)
RM_X := ( INT_TO_REAL ( RM_Y ) * m + b);			(*Geradengleichung*)
IF (RM_X < Y_UG) OR (RM_X <= 2)  THEN
	RM_X := Y_UG;
END_IF;
IF (RM_X > Y_OG) OR (RM_X >= 98)  THEN
	RM_X := Y_OG;
END_IF;

(*Auswertung Rückmeldefehler*)
BereichOG :=  Yx + ((Y_OG - Y_UG) * 0.20);
BereichUG :=  Yx -  ((Y_OG - Y_UG) * 0.20);
RMF(IN:=(((BereichOG < RM_X OR BereichUG > RM_X) AND DDC) OR Stoe_Rmx) AND NOT QuittRMF, PT:=T_RM);
Stoe_Rmx := RMF.Q;

(*Auswertung Störung Frost*)
Stoe_Frostx := (NOT Frost);

(*Auswertung Störung*)
Maske := Konfig AND 2#00001000;
IF Maske = 8 THEN
	SAx := Stoe_Rmx ;
	ELSE	SAx := Stoe_Rmx;
END_IF;

(*Quittierung Rückmeldefehler*)
QuittRMF := FALSE;
Maske := Konfig AND 2#00000001;
IF Maske = 1 THEN
	IF ((BereichOG > RM_X AND BereichUG < RM_X)) AND Stoe_Rmx AND Quitt THEN
		QuittRMF := TRUE;
	END_IF;
	ELSE IF Stoe_Rmx AND Quitt THEN
		QuittRMF := TRUE;
	END_IF;
END_IF;

(*Ansteuerung Antrieb*)
IF FRG AND DDC THEN
	m := ((Y_OG - Y_UG) / 100);	(*Steigung*)
	b := Y_UG;					(*Nulldurchgang*)
	Yx := m * Auto_Stell + b;		(*Geradengleichung*)
	IF TA_Gx OR TA_Vx THEN
		Maske := 2#00000001;
		IF V_STELL > Y_OG THEN
			V_STELL := Y_OG;
		END_IF;
		IF V_STELL < Y_UG THEN
			V_STELL := Y_UG;
		END_IF;
		Yx := V_STELL;
	END_IF;
	IF TA_Px THEN
		IF P_STELL > Y_OG THEN
			P_STELL := Y_OG;
		END_IF;
		IF P_STELL < Y_UG THEN
			P_STELL := Y_UG;
		END_IF;
		Yx := P_STELL;
	END_IF;
	IF Stoe_Rmx THEN	(*Bei Rückmeldefehler Antrieb = Ein || Antrieb = Aus || Antrieb = Auto*)
		Maske := Konfig AND 2#00000110;
		IF Maske = 4 THEN
			Yx := Yx;
			ELSE IF Maske = 2 THEN
				Yx := Y_OG;
				ELSE
					Yx := Y_UG;
			END_IF;
		END_IF;
	END_IF;

	(*Blockierschutz*)
	TON_BLOCK (IN:= BLOCK AND ( Y = Y_UG), PT:=T_BLOCK);
	TP_BLOCK (IN:= TON_BLOCK.Q, PT:= T#5m);
	IF TP_BLOCK.Q THEN
		Yx := Y_OG;
	END_IF;
	BLOCK_EIN := TP_BLOCK.Q;
ELSE
	Yx := Y_UG;
END_IF;

IF Stoe_Frostx AND DDC THEN
	Yx := Y_OG;
END_IF;

(*Skalierung Ansteuerung*)
IF  (Y_OG - Y_UG) = 0 THEN
    Y_OUT := 0;                                    (*DIV / NULL*)
    ELSE
        m := (32767 / (Y_OG - Y_UG));            (*Steigung*)
        b := Y_UG * m * -1;                        (*Nulldurchgang*)
        Y_OUT := REAL_TO_INT (m * Yx + b);    (*Geradengleichung*)

	(*Ansteuerung gegenläufig*)
	Maske := Konfig AND 2#01000000;
	IF Maske = 64 THEN
		m :=-1;	(*Steigung*)
		b := 32767;
		Y_OUT :=REAL_TO_INT( INT_TO_REAL (Y_OUT) * m + b);
	END_IF;

	(*Ansteuerung 2-10V*)
	Maske := Konfig AND 2#00100000;
	IF Maske = 32 THEN
		m :=0.8;	(*Steigung*)
		b := 0.2 * 32767;
		Y_OUT :=REAL_TO_INT( INT_TO_REAL (Y_OUT) * m + b);
	END_IF;
END_IF;

IF Yx > 97 THEN
Y := 100;
ELSE
Y := Yx;
END_IF

IF Yx < 2 THEN
Y := 0;
ELSE
Y := Yx;
END_IF




(*Meldeunterdrückung*)
U_IO_Verz(IN:=U_IO, PT:=T#5s);
U_IO_X := U_IO_Verz.Q;
IF U_IO_X THEN
	NOTB	:=	NOTBx	;
	TA_P	:=	TA_Px	;
	TA_V	:=	TA_Vx	;
	TA_G	:=	TA_Gx	;
	S_TA	:=	S_TAx	;
	STOE_RM	:=	STOE_RMx	;
 	STOE_FROST	:=	Stoe_Frostx;
	SA	:=	SAx	;
END_IF;

Sperre:=NOT FRG;

END_FUNCTION_BLOCK

// ---- MRA/02_FUNKTIONS_BAUSTEINE/BUS/KNX/KNX_BOOL_READ_WRITE.TcPOU
FUNCTION_BLOCK KNX_BOOL_READ_WRITE
VAR_INPUT
	BOOL_IN : BOOL;
	GRUPPEN_ADRESSE_IN : STRING;
	GRUPPEN_ADRESSE_OUT : STRING;
	EIB_DATA_st : Tc2_EIB.EIB_REC;
END_VAR

VAR_OUTPUT
 	BOOL_OUT : BOOL;
END_VAR
VAR
EIB_BIT_SEND : EIB_BIT_SEND;
EIB_BIT_REC : EIB_BIT_REC;
END_VAR

EIB_BIT_SEND(
	Group_Address:= STRING_TO_EIB_GRP_ADDR(GRUPPENADRESSE:= GRUPPEN_ADRESSE_IN ), 
	bData:= BOOL_IN, 
	str_Rec:= EIB_DATA_st, 
	bError=> , 
	iErrorID=> );
	
EIB_BIT_REC(
	Group_Address:= STRING_TO_EIB_GRP_ADDR(GRUPPENADRESSE:= GRUPPEN_ADRESSE_OUT ),
 	strData_Rec:= EIB_DATA_st,
 	bDataReceive=>  ,
 	bData=> BOOL_OUT);

END_FUNCTION_BLOCK

// ---- MRA/02_FUNKTIONS_BAUSTEINE/BUS/KNX/KNX_REAL_READ_WRITE.TcPOU
FUNCTION_BLOCK KNX_REAL_READ_WRITE
VAR_INPUT
	
GRUPPENADRESSE	:	STRING;
KNX_STRUCTUR	:	EIB_REC;
REAL_IN			:	REAL;
END_VAR
VAR_OUTPUT
REAL_OUT		:	REAL;	
INFO			:	STRING;
ERROR_OUT		:	BOOL;
END_VAR
VAR
KNX_2BYTE_TO_REAL	: EIB_2OCTET_FLOAT_REC;
STARTUP_READ		: EIB_READ_SEND;
EIB_ERROR			: INT;
EIB_ADRESSE			: Tc2_EIB.EIB_GROUP_ADDR;	
TON_KALTSTART 		: Tc2_Standard.TON;
R_TRIG_STARTUP_READ	: R_TRIG;

EIB_2OCTET_FLOAT_SEND : EIB_2OCTET_FLOAT_SEND;
END_VAR


TON_KALTSTART(IN := TRUE, PT := T#10S);
R_TRIG_STARTUP_READ(CLK := TON_KALTSTART.Q);

EIB_ADRESSE := STRING_TO_EIB_GRP_ADDR(GRUPPENADRESSE := GRUPPENADRESSE);


STARTUP_READ(Group_Address:= EIB_ADRESSE , 
	         bRead:=   R_TRIG_STARTUP_READ.Q, 
	         str_Rec:= KNX_STRUCTUR , 
	         iErrorID=> EIB_ERROR , 
	        );
			
CASE EIB_ERROR OF	
	0			: INFO := 	'NO_EIB_ERROR'                       ;
	1			: INFO := 	'WRONG_EIB_PHYS_ADDR'                ;
	2			: INFO := 	'WRONG_EIB_GROUP_ADDR'               ;
	3			: INFO := 	'WRONG_EIB_GROUP_LEN'                ;
	4			: INFO := 	'WRONG_EIB_NO_FILTER'                ;
	10			: INFO := 	'WRONG_EIB_FIRMWARE'                 ;
	11			: INFO := 	'WRONG_EIB_MODE'                     ;
	12			: INFO := 	'WRONG_MODE'                         ;
	14			: INFO := 	'WRONG_EIB_FIRMWARE_B1_NECESSARY'    ;
	15			: INFO := 	'WRONG_EIB_FIRMWARE_B3_NECESSARY'    ;
	20			: INFO := 	'WRONG_EIB_DATA_LEN'                 ;
	21			: INFO := 	'ERROR_EIB_SERVICE_NOT_SUPPORT'      ;
	30			: INFO := 	'KL6301_TP_TOGGLE_ERROR'             ;
	31			: INFO := 	'TIME_OUT'                           ;
	32			: INFO := 	'KL6301_NO_RESPONSE_FROM_TERMINAL'   ;
	40			: INFO := 	'ERROR_SEND_8BIT_WRONG_Scaling_Mode' ;
	100			: INFO := 	'ERROR_EIB_PHY_ADDR_NOT_SUPPORT'     ;
	101			: INFO := 	'ERROR_EIB_WRITE_DATA'               ;
	102			: INFO := 	'MONITOR_MODE_LEN_IS_NOT_OK_MUST_0'  ;
	103			: INFO := 	'MONITOR_MODE_ADDR_IS_NOT_OK_MUST_0' ;
	104			: INFO := 	'WATCHDOG_ERROR_NO_SEND'             ;
	16#0BBB		: INFO := 	'ERROR_EIB_NO_ACK'                   ;
	16#FAFB		: INFO := 	'ERROR_EIB_NO_COM_TO_TP'             ;
	16#0FCC		: INFO := 	'ERROR_TP_TEMP_WARNING'              ;
	16#17CC		: INFO := 	'ERROR_TP_PROTOCOL_ERROR'            ;
	16#27CC		: INFO := 	'ERROR_TP_TRANSMITTER_ERROR'         ;
	16#47CC		: INFO := 	'ERROR_TP_RECEIVE_ERROR'             ;
	16#87CC		: INFO := 	'ERROR_TP_SLAVE_COLLISION'           ;	
END_CASE



(*KNX_2BYTE_TO_REAL(Group_Address:= EIB_ADRESSE,
 				  strData_Rec:= KNX_STRUCTUR,
				  rData => REAL_OUT);*)

IF ADR(REAL_OUT) <> ADR(REAL_IN) THEN
	
	EIB_2OCTET_FLOAT_SEND(
				  Group_Address:= EIB_ADRESSE, 
	              rData:= REAL_IN, 
	              str_Rec:= KNX_STRUCTUR, 
	              iErrorID=> EIB_ERROR);
	REAL_OUT := REAL_IN;
END_IF
				  

				  
			
IF EIB_ERROR > 0 THEN
ERROR_OUT := TRUE;

ELSE
ERROR_OUT := FALSE;	

END_IF

END_FUNCTION_BLOCK

// ---- MRA/02_FUNKTIONS_BAUSTEINE/BUS/ModBus/FB_MODBUS_DEVICE.TcPOU
FUNCTION_BLOCK FB_MODBUS_DEVICE
VAR_INPUT
	fbMaster					: ITF_MODBUS_RTU;
	bEnable						: BOOL;
	// Modbus device address
	nUnitAddr					: BYTE;
END_VAR
VAR_OUTPUT
	bBusy						: BOOL;
	bError						: BOOL;
	eError						: Tc2_ModbusRTU.MODBUS_ERRORS;
	rTemperature1: REAL;
	rHumdity1: REAL;
	rTemperature2: REAL;
	rHumdity2: REAL;
END_VAR
VAR
	fbRtrigUnitAddr				: R_TRIG;
	nWriteOutputRegsM			: INT;
	nReadReg					: ARRAY [0..3] OF WORD;

END_VAR

fbRtrigUnitAddr(CLK:= bEnable AND nUnitAddr = fbMaster.nCurrentUnitAddr );
IF bEnable THEN
	IF fbRtrigUnitAddr.Q THEN
		bBusy := TRUE;
		// ###############################
		// Insert here the Modbus Commands
		// ###############################
	
		fbMaster.mAddRequest(nUnitAddr := nUnitAddr, nRegModbusAddr := 0, nFunction := E_MODBUS_FUNCTION.Read_Holding_Registers, pVar := ADR(nReadReg), nSizeOfVar := SIZEOF(nReadReg), pError := ADR(eError));
		
		// ###############################
		// End of Modbus Commands
		// ###############################
	ELSE
		IF fbMaster.nRequestNo = 0 THEN
			bBusy :=FALSE;
		END_IF
	END_IF
	bError := eError <> Tc2_ModbusRTU.MODBUS_ERRORS.MODBUSERROR_NO_ERROR;
ELSE
	bBusy := FALSE;
	bError := FALSE;
	eError := Tc2_ModbusRTU.MODBUS_ERRORS.MODBUSERROR_NO_ERROR;
END_IF

rTemperature1 := TO_REAL(nReadReg[0])/10.0;
rHumdity1 :=  TO_REAL(nReadReg[1])/10.0;
rTemperature2 := TO_REAL(nReadReg[2])/10.0;
rHumdity2 :=  TO_REAL(nReadReg[3])/10.0;

END_FUNCTION_BLOCK

// ---- MRA/02_FUNKTIONS_BAUSTEINE/MASCHIENENBAU/fb_Drehzahl.TcPOU
FUNCTION_BLOCK fb_Drehzahl
VAR_INPUT

		TRIGGER : BOOL;	

END_VAR
VAR_OUTPUT
	
	UMDREHUNGEN_PRO_MINUTE : INT;
	
END_VAR
VAR
	
		
	R_TRIG: R_TRIG;
	TON_COUNTER : TON;
	DREHIMPULSE_1S : INT;

END_VAR

R_TRIG(CLK:= TRIGGER);

TON_COUNTER(IN:= NOT TON_COUNTER.Q, PT := T#5S);


IF R_TRIG.Q THEN
	

	DREHIMPULSE_1S := DREHIMPULSE_1S + 1;

END_IF

IF TON_COUNTER.Q THEN
	

	UMDREHUNGEN_PRO_MINUTE := DREHIMPULSE_1S * 12;
	DREHIMPULSE_1S := 0;

END_IF

END_FUNCTION_BLOCK

// ---- MRA/02_FUNKTIONS_BAUSTEINE/Testing/Aggregate/fb_IBN_Pumpe.TcPOU
FUNCTION_BLOCK fb_IBN_Pumpe
VAR_INPUT
	AUTO_EIN : BOOL; //Ansteuerung Auf
	LOGGING_NAME : STRING; //Name des Ventil für den Log Eintrag
	TIME_STAMP : STRING; //Zeitstempell für den Log Eintrag
	MAX_LOGG_ENTRY : INT := 10000;
END_VAR
VAR_OUTPUT
	RM : BOOL; //Rückmeldung 
END_VAR
VAR_IN_OUT
	LOGGING_ENTRY : INT; //Hier einen Integer verlinken auf dem die Log Positioon gelesen und dann erhöht wird, muss mit allen anderen FB's mit Log verdunden werden
	LOGGING_MESSAGE : STRING; //Hier ein beliebig Großese String Array Verlinken und den Logg Entry alls Array Position angeben , muss mit allen anderen FB's mit Log verdunden werden
END_VAR
VAR
	TON_EIN : Tc2_Standard.TON;
	TON_AUS : Tc2_Standard.TON;
	F_TRIG_RM_ZU: F_TRIG;
	R_TRIG_RM_AUF: R_TRIG;
	BUFFER_STRING : STRING;
END_VAR




IF AUTO_EIN THEN
	//Rückmeldung 	

	TON_AUS(IN := FALSE);
	
	TON_EIN(IN := TRUE, PT := T#5S);	
	RM := TON_EIN.Q ;
	
	//LOG	
	R_TRIG_RM_AUF(CLK := RM);
	
	IF R_TRIG_RM_AUF.Q THEN
		LOGGING_ENTRY := LOGGING_ENTRY + 1;
 		BUFFER_STRING := Tc2_Standard.CONCAT( LOGGING_NAME , ' Rückmeldung Ein   TIME:');
		LOGGING_MESSAGE := CONCAT(BUFFER_STRING , TIME_STAMP);
	END_IF
	
ELSE
	//Rückmeldung 	

	TON_EIN(IN := FALSE);
	
	TON_AUS(IN := TRUE, PT := T#5S);
	RM := NOT TON_AUS.Q ;	
	
	//LOG	
	F_TRIG_RM_ZU(CLK := RM);
	
	IF F_TRIG_RM_ZU.Q THEN
		LOGGING_ENTRY := LOGGING_ENTRY + 1;
		BUFFER_STRING := Tc2_Standard.CONCAT( LOGGING_NAME , ' Rückmeldung Aus   TIME:');
		LOGGING_MESSAGE := CONCAT(BUFFER_STRING , TIME_STAMP);	END_IF

END_IF




IF LOGGING_ENTRY = MAX_LOGG_ENTRY THEN
	LOGGING_ENTRY := 1;
END_IF

END_FUNCTION_BLOCK

// ---- MRA/02_FUNKTIONS_BAUSTEINE/Testing/Aggregate/fb_IBN_Ventil.TcPOU
FUNCTION_BLOCK fb_IBN_Ventil //Zum Simmuliern eine Ventils
VAR_INPUT
	AUTO_AUF : BOOL; //Ansteuerung Auf
	LOGGING_NAME : STRING; //Name des Ventil für den Log Eintrag
	TIME_STAMP : STRING; //Zeitstempell für den Log Eintrag
	MAX_LOGG_ENTRY : INT := 10000;
END_VAR
VAR_OUTPUT
	RM_AUF : BOOL; //Rückmeldung offen des Ventil
	RM_ZU  : BOOL; //Rückmeldung geschlossen des Ventil
END_VAR
VAR_IN_OUT
	LOGGING_ENTRY : INT; //Hier einen Integer verlinken auf dem die Log Positioon gelesen und dann erhöht wird, muss mit allen anderen FB's mit Log verdunden werden,
	LOGGING_MESSAGE : STRING; //Hier ein beliebig Großese String Array Verlinken und den Logg Entry alls Array Position angeben , muss mit allen anderen FB's mit Log verdunden werden
END_VAR
VAR
	TON_AUF : Tc2_Standard.TON;
	TON_ZU 	: Tc2_Standard.TON;
	R_TRIG_RM_ZU: Tc2_Standard.R_TRIG;
	R_TRIG_RM_AUF: Tc2_Standard.R_TRIG;
	BUFFER_STRING : STRING;
 
END_VAR

IF AUTO_AUF THEN
	//Rückmeldung 	
	RM_ZU := FALSE;	
	TON_ZU(IN := FALSE);
	
	TON_AUF(IN := NOT RM_ZU, PT := T#5S);	
	RM_AUF := TON_AUF.Q ;
	
	//LOG	
	R_TRIG_RM_AUF(CLK := RM_AUF);
	
	IF R_TRIG_RM_AUF.Q THEN
		LOGGING_ENTRY := LOGGING_ENTRY + 1;
		BUFFER_STRING := Tc2_Standard.CONCAT( LOGGING_NAME , ' Rückmeldung offen   		TIME:');
		LOGGING_MESSAGE := CONCAT(BUFFER_STRING , TIME_STAMP);
	END_IF
	
ELSE
	//Rückmeldung 	
	RM_AUF := FALSE;	
	TON_AUF(IN := FALSE);
	
	TON_ZU(IN := NOT RM_AUF, PT := T#5S);
	RM_ZU := TON_ZU.Q ;	
	
	R_TRIG_RM_ZU(CLK := RM_ZU);
	
	IF R_TRIG_RM_ZU.Q THEN
		LOGGING_ENTRY := LOGGING_ENTRY + 1;
		BUFFER_STRING := Tc2_Standard.CONCAT( LOGGING_NAME , ' Rückmeldung geschlossen   		TIME:');
		LOGGING_MESSAGE := CONCAT(BUFFER_STRING , TIME_STAMP);
	END_IF

END_IF

IF LOGGING_ENTRY = MAX_LOGG_ENTRY THEN
	LOGGING_ENTRY := 1;
END_IF

END_FUNCTION_BLOCK

// ---- MRA/02_FUNKTIONS_BAUSTEINE/Testing/Aggregate/fb_IBN_Ventil_ohne_Log.TcPOU
FUNCTION_BLOCK fb_IBN_Ventil_ohne_Log
VAR_INPUT
	AUTO_AUF : BOOL;
	VERFAHRZEIT : TIME;
END_VAR
VAR_OUTPUT
	RM_AUF : BOOL;
	RM_ZU  : BOOL;
END_VAR
VAR
	TON_AUF : Tc2_Standard.TON;
	TON_ZU 	: Tc2_Standard.TON;
END_VAR

	
IF AUTO_AUF THEN
	//Rückmeldung 	
	RM_ZU := FALSE;	
	TON_ZU(IN := FALSE);
	
	TON_AUF(IN := NOT RM_ZU, PT := VERFAHRZEIT);	
	RM_AUF := TON_AUF.Q ;	
ELSE
	//Rückmeldung 	
	RM_AUF := FALSE;	
	TON_AUF(IN := FALSE);
	
	TON_ZU(IN := NOT RM_AUF, PT := VERFAHRZEIT);
	RM_ZU := TON_ZU.Q ;	

END_IF

END_FUNCTION_BLOCK

// ---- MRA/02_FUNKTIONS_BAUSTEINE/Testing/fb_Log.TcPOU
FUNCTION_BLOCK fb_Log
VAR_INPUT
		INPUT_STRING: STRING;
		SYSTEM_TIME : STRING;
		CLEAR_LOGG_ARRAY: BOOL;
END_VAR
VAR_IN_OUT
		LOGG_ENTRY    : INT;
		logging_array : ARRAY [1..1000] OF STRING(500);
END_VAR
VAR
		INPUT_STRING_BUFFER: STRING;
		clear_loggarray: ARRAY [1..1000] OF STRING(500);
		BUFFER_STRING: STRING(500);
END_VAR

	IF INPUT_STRING <> INPUT_STRING_BUFFER THEN
	 	INPUT_STRING_BUFFER :=	INPUT_STRING;
		LOGG_ENTRY := LOGG_ENTRY + 1;
		IF LOGG_ENTRY > 999 THEN
			LOGG_ENTRY := 0;
		END_IF
		BUFFER_STRING := CONCAT('      TIME STAMP:  ', SYSTEM_TIME );
		LOGGING_ARRAY[LOGG_ENTRY] := CONCAT(INPUT_STRING, BUFFER_STRING );		
	END_IF

	IF CLEAR_LOGG_ARRAY THEN
		Tc2_System.MEMCPY(destAddr:=ADR(logging_array) , srcAddr:=ADR(clear_loggarray) , n:=SIZEOF(logging_array));
		logg_entry := 0;
	END_IF

END_FUNCTION_BLOCK

// ---- MRA/02_FUNKTIONS_BAUSTEINE/Visualisierung/fb_Zeitprogramm.TcPOU
FUNCTION_BLOCK fb_Zeitprogramm 
VAR_INPUT
	FREIGABE 							: BOOL;
	START_UHRZEIT						: STRING;     //Format Info: '12:12'
	START_DATUM							: STRING;	 //Format Info: '01.11'
	END_UHRZEIT							: STRING;     //Format Info: '12:12'
	END_DATUM							: STRING;	 //Format Info: '01.11'	
END_VAR
VAR_OUTPUT
	ZEITPROGRAMM_AKTIV					: BOOL;
END_VAR
VAR			  
	AKTUELLE_STUNDE						: WORD;
	AKTUELLE_MINUTE		 				: WORD;
	AKUTELLE_SEKLUNDE					: WORD; 	
	AKTUELLES_JAHR		  				: WORD;   	
	AKTUELLER_MONAT		 				: WORD;  	
	AKTUELLER_TAG		   				: WORD;
	
	START_MINUTE						: WORD;
	START_STUNDE						: WORD;
	START_TAG							: WORD;
	START_MONAT							: WORD;
	
	END_MINUTE							: WORD;
	END_STUNDE							: WORD;
	END_TAG								: WORD;
	END_MONAT							: WORD;

	
	
	
	
	state								: INT;
	R_TRIG_FREIGABE						: R_TRIG;
	AMS_NET_ID 							: STRING;
	ADS_TIME							: Tc2_Utilities.NT_GetTime;
	GET_AMS_NET_ID						: Tc2_Utilities.FB_GetLocalAmsNetId;
	st_ADS_TIME							: Tc2_Utilities.TIMESTRUCT;
	lese_interval						: TOF;
END_VAR

lese_interval(	PT	:=	T#1200MS,	IN	:=	NOT	lese_interval.Q	);

GET_AMS_NET_ID(	bExecute:= TRUE , 	AddrString=> AMS_NET_ID); 

ADS_TIME(
	NETID:= AMS_NET_ID, 
	START:= lese_interval.Q, 	
	TIMESTR=> st_ADS_TIME );	
	
	AKTUELLE_STUNDE 	 	:= st_ADS_TIME.wHour;
	AKTUELLE_MINUTE		  	:= st_ADS_TIME.wMinute;
	AKUTELLE_SEKLUNDE		:= st_ADS_TIME.wSecond;
	AKTUELLES_JAHR		  	:= st_ADS_TIME.wYear;
	AKTUELLER_MONAT		 	:= st_ADS_TIME.wMonth;
	AKTUELLER_TAG     		:= st_ADS_TIME.wDay;

	START_TAG				:= STRING_TO_WORD(Tc2_Standard.LEFT(START_DATUM, 2));
	START_MONAT				:= STRING_TO_WORD(Tc2_Standard.RIGHT(START_DATUM, 2));
	
	START_STUNDE			:= STRING_TO_WORD(Tc2_Standard.LEFT(START_UHRZEIT, 2));
	START_MINUTE			:= STRING_TO_WORD(Tc2_Standard.RIGHT(START_UHRZEIT, 2));
	
	END_TAG					:= STRING_TO_WORD(Tc2_Standard.LEFT(END_DATUM, 2));
	END_MONAT				:= STRING_TO_WORD(Tc2_Standard.RIGHT(END_DATUM, 2));
	
	END_STUNDE				:= STRING_TO_WORD(Tc2_Standard.LEFT(END_UHRZEIT, 2));
	END_MINUTE				:= STRING_TO_WORD(Tc2_Standard.RIGHT(END_UHRZEIT, 2));
	
R_TRIG_FREIGABE(CLK := FREIGABE);

IF R_TRIG_FREIGABE.Q THEN state := 1; END_IF

CASE state OF
	
	0: 
		ZEITPROGRAMM_AKTIV := FALSE;
		
	1:
		IF (START_MONAT <= AKTUELLER_MONAT) AND (END_MONAT >= AKTUELLER_MONAT) THEN
			state := 2;
		ELSE
			state := 6;
		END_IF
		
	2: 	
		IF (START_TAG <= AKTUELLER_TAG) AND (END_TAG >= AKTUELLER_TAG) THEN
			state := 3;		
		ELSE
			state := 6;
		END_IF	
		
	3:
		IF (START_STUNDE <= AKTUELLE_STUNDE) AND (END_STUNDE >= AKTUELLE_STUNDE) THEN
			state := 4;		
		ELSE
			state := 6;
		END_IF
		
	4:
		IF (START_MINUTE = AKTUELLE_MINUTE) AND (START_STUNDE = AKTUELLE_STUNDE)  THEN
			ZEITPROGRAMM_AKTIV := TRUE;
		ELSIF (END_MINUTE = AKTUELLE_MINUTE) AND (END_STUNDE = AKTUELLE_STUNDE)  THEN
			ZEITPROGRAMM_AKTIV := FALSE;		
		END_IF	
	6:
		ZEITPROGRAMM_AKTIV := FALSE;
		state := 1;

		

END_CASE

END_FUNCTION_BLOCK

// ---- MRA/03_BSP_PRG/06_KNX/KNX.TcPOU
PROGRAM KNX
VAR
	KL6301: KL6301;
	

bActivate        : BOOL;
idx              : INT := 1;
EIB_PHYS_ADDR    : EIB_PHYS_ADDR;
EIB_GROUP_FILTER : ARRAY [1..8] OF EIB_GROUP_FILTER;
iMode            : INT;
tTimeout         : TIME := T#10S;

	
bActive      : BOOL;
bReady       : BOOL;
bError       : BOOL;
iErrorId     : EIB_Error_Code;
	fbWait: TON;
	bActivateTest: BOOL := TRUE;
	fbRtrigReady: R_TRIG;
	TEST1: BOOL;
END_VAR

(* ##################################################################################################################### *)
(* Definition der physikalischen Adresse jeder Klemme *)
	(* Adresse kann nur an eine Klemme vergeben werden *)

	EIB_PHYS_ADDR.Area		:= 1;
	EIB_PHYS_ADDR.Line		:= 7;
	EIB_PHYS_ADDR.Device	:= 200;


(* ##################################################################################################################### *)
(* Bus - Filter für die Gruppenadressen [max. 8] *)

	(* Filter 1	*)
		EIB_GROUP_FILTER[1].GROUP_ADDR.MAIN 	:= 0;
		EIB_GROUP_FILTER[1].GROUP_ADDR.SUB_MAIN	:= 6;
		EIB_GROUP_FILTER[1].GROUP_ADDR.NUMBER	:= 0;
		EIB_GROUP_FILTER[1].GROUP_LEN			:= 63;
	(* Filter 2	*)
		EIB_GROUP_FILTER[2].GROUP_ADDR.MAIN 	:= 0;
		EIB_GROUP_FILTER[2].GROUP_ADDR.SUB_MAIN	:= 6;
		EIB_GROUP_FILTER[2].GROUP_ADDR.NUMBER	:= 64;
		EIB_GROUP_FILTER[2].GROUP_LEN			:= 63;
	(* Filter 3	*)
		EIB_GROUP_FILTER[3].GROUP_ADDR.MAIN 	:= 0;
		EIB_GROUP_FILTER[3].GROUP_ADDR.SUB_MAIN	:= 6;
		EIB_GROUP_FILTER[3].GROUP_ADDR.NUMBER	:= 128;
		EIB_GROUP_FILTER[3].GROUP_LEN			:= 63;
	(* Filter 4	*)
		EIB_GROUP_FILTER[4].GROUP_ADDR.MAIN 	:= 0;
		EIB_GROUP_FILTER[4].GROUP_ADDR.SUB_MAIN	:= 6;
		EIB_GROUP_FILTER[4].GROUP_ADDR.NUMBER	:= 192;
		EIB_GROUP_FILTER[4].GROUP_LEN			:= 63;

fbWait(IN:= Allgemein.CX_Status = 0, PT:= T#100MS);

KL6301(
	bActivate:= fbWait.Q,
	idx:= idx, 
	EIB_PHYS_ADDR:= EIB_PHYS_ADDR, 
	EIB_GROUP_FILTER:=EIB_GROUP_FILTER , 
	iMode:=iMode , 
	tTimeout:=tTimeout , 
	bActive=> bActive, 
	bReady=> bReady, 
	bError=> bError, 
	iErrorId=>iErrorId , 
	str_Data_Rec=> str_Data_Rec, 
	KL6301_IN:=KL6301_IN , 
	KL6301_OUT:=KL6301_OUT );


	
	


	


	

IF bReady THEN	
	KNX_BOOL_SEND(GRUPPENADRESSE:='0.6.0' , KNX_STRUCTUR:= str_Data_Rec , REAL_OUT=>KNX_E01_Putzraum_Temperatur, INFO=> ERROR_INFO[1] ,	ERROR_OUT=>KNX_E01_Putzraum_Temperatur_SS01);

 END_IF

END_PROGRAM

// ---- MRA/04_RRVALUE/fb_REAL_RRVALUE.TcPOU
FUNCTION_BLOCK fb_REAL_RRVALUE
VAR_INPUT
EIB_DATA_st : Tc2_EIB.EIB_REC;
END_VAR
VAR_IN_OUT
st_REAL_RRVALUE : st_REAL_RRVALUE;	
END_VAR
VAR
	TON_KALTSTART : Tc2_Standard.TON;
	

	//Skallierung
	i_r_in		:REAL;
	i_r_x_min	:REAL;
	i_r_x_max	:REAL;
	i_r_y_min	:REAL;
	i_r_y_max	:REAL;
	
	//Grenzwert
	TON_MAX_VALUE : Tc2_Standard.TON;
	TON_MIN_VALUE : Tc2_Standard.TON;
	
	//KNX
	EIB_2OCTET_FLOAT_SEND : TC2_EIB.EIB_2OCTET_FLOAT_SEND;
	EIB_2OCTET_FLOAT_REC : Tc2_EIB.EIB_2OCTET_FLOAT_REC;	
	EIB_READ_SEND: EIB_READ_SEND;
END_VAR

TON_KALTSTART(IN := TRUE, PT:= T#10s);

a_scal();
a_minmax();
a_knx();

ACTION a_knx:
IF st_REAL_RRVALUE.b_KNX_Enable THEN	
		
			
		EIB_READ_SEND(
			Group_Address:= STRING_TO_EIB_GRP_ADDR(GRUPPENADRESSE:= st_REAL_RRVALUE.s_KNX_Addres  ) , 
			bRead:= TON_KALTSTART.Q, 
			str_Rec:= EIB_DATA_st); 
		
		


		IF st_REAL_RRVALUE.b_KNX_Write_Mode THEN
			
			EIB_2OCTET_FLOAT_SEND(
				Group_Address:= STRING_TO_EIB_GRP_ADDR(GRUPPENADRESSE:= st_REAL_RRVALUE.s_KNX_Addres  ) , 
				rData:= st_REAL_RRVALUE.r_in_Value, 
				str_Rec:= EIB_DATA_st);
		
		ELSE
		
			EIB_2OCTET_FLOAT_REC(
				Group_Address:= STRING_TO_EIB_GRP_ADDR(GRUPPENADRESSE:= st_REAL_RRVALUE.s_KNX_Addres ) , 
				strData_Rec:= EIB_DATA_st, 
				rData=> st_REAL_RRVALUE.r_in_Value);		
		
		END_IF

END_IF
END_ACTION

ACTION a_minmax:
//Grenzwert
IF st_REAL_RRVALUE.b_Enable_MinMax THEN
	
	//Grenzwert Oben
	TON_MAX_VALUE(IN:= st_REAL_RRVALUE.r_out_Value >= st_REAL_RRVALUE.r_MaxValue, PT := TO_TIME(st_REAL_RRVALUE.t_MinMax_Delay * 1000));
	
	IF TON_MAX_VALUE.Q THEN
		st_REAL_RRVALUE.b_MaxValue_Reached := TRUE;
	ELSE
		st_REAL_RRVALUE.b_MaxValue_Reached := FALSE;
	END_IF
	
	
	//Grenzwert Unten	
	TON_MIN_VALUE(IN:= st_REAL_RRVALUE.r_out_Value <= st_REAL_RRVALUE.r_MinValue, PT := TO_TIME(st_REAL_RRVALUE.t_MinMax_Delay * 1000));
	
	IF TON_MIN_VALUE.Q THEN
		st_REAL_RRVALUE.b_MinValue_Reached := TRUE;
	ELSE
		st_REAL_RRVALUE.b_MinValue_Reached := FALSE;
	END_IF
	
	
	
ELSE
	
	st_REAL_RRVALUE.b_MinValue_Reached := FALSE;
	st_REAL_RRVALUE.b_MaxValue_Reached := FALSE;

END_IF
END_ACTION

ACTION a_scal:

END_ACTION

END_FUNCTION_BLOCK
